// TwinCAT 3 PLC project RFID_lib
// Title: RFID_Sensor
// Company: Thomas More
// Author: Arno Joosen
// ProjectVersion: 0.0.4
// ProgramVersion: 3.1.4023.0
// libraries:
//   Buffer Lib, * (Thomas More)
//   RFID universal data interface TwinCAT, * (Turck)
//   Tc2_Standard, * (Beckhoff Automation GmbH)
//   Tc2_System, * (Beckhoff Automation GmbH)
//   Tc3_Module, * (Beckhoff Automation GmbH)
// project tree:
//   DUTs/ Read_State.TcDUT, RFID_Sensor.TcDUT, RFID_SensorState.TcDUT, RFID_Error.TcDUT, RFID_Tag_Data.TcDUT, Tag_UID.TcDUT, Wread_State.TcDUT
//   POUs/ ID_equal_to_ID.TcPOU, RFID_Sensor_Read.TcPOU, RFID_Sensor_Wread.TcPOU, RFID_Update.TcPOU
//   POUs/Read_Tag_Data/ RFID_Get_Bool.TcPOU, RFID_Get_Int.TcPOU, RFID_Get_Real.TcPOU, RFID_Get_String.TcPOU
//   POUs/Wread_Tag_Data/ RFID_Set_Bool.TcPOU, RFID_Set_Int.TcPOU, RFID_Set_Real.TcPOU, RFID_Set_String.TcPOU
//   Version/ Global_Version.TcGVL
// real-time tasks:
//   TASK PlcTask: cycle T#10ms, priority 20, ADS port 350
//   TASK PlcTask1: cycle T#10ms, priority 21, ADS port 351
//   TASK PlcTask2: cycle T#10ms, priority 22, ADS port 352
//   TASK PlcTask3: cycle T#10ms, priority 23, ADS port 353

// ---- DUTs/Read_State.TcDUT
{attribute 'qualified_only'}
{attribute 'strict'}
TYPE Read_State :
(
	Triggerd := 0,
	DataWritten := 1,
	Done := 2
)UINT;
END_TYPE

// ---- DUTs/RFID_Sensor.TcDUT
TYPE RFID_Sensor :
STRUCT
	Input AT %I* : CompactInput_t;
	Ouput AT %Q* : CompactOutput_t;
	
	Input_Buffer AT %I* : ARRAY[0..127] OF BYTE;
	Output_Buffer AT %Q* : ARRAY[0..127] OF BYTE;
	
	TxBuffer : ARRAY[0..127] OF BYTE;
	
	State : RFID_SensorState := RFID_SensorState.idel;
	ReadState : Read_State;
	WreadState : Wread_State;
	Pagina : UINT;
	CurrentTagData : RFID_Tag_Data;
END_STRUCT
END_TYPE

// ---- DUTs/RFID_SensorState.TcDUT
{attribute 'qualified_only'}
{attribute 'strict'}
TYPE RFID_SensorState :
(
	idel := 0,
	ReadTag := 1,
	WreadTag := 2,
	Error := 3
) UINT;
END_TYPE

// ---- DUTs/RFID_Error.TcDUT
{attribute 'qualified_only'}
{attribute 'strict'}
TYPE RFID_Error :
(
	None := 0,
	Not_Connected := 1,
	Time_Out := 2,
	Sesnor := 3
) UINT;
END_TYPE

// ---- DUTs/RFID_Tag_Data.TcDUT
TYPE RFID_Tag_Data :
STRUCT
	Data : ARRAY[0..127] OF BYTE;
	UID : Tag_UID;
	Layout : Buffer_Layout;
END_STRUCT
END_TYPE

// ---- DUTs/Tag_UID.TcDUT
TYPE Tag_UID : ARRAY[0..7] OF USINT; END_TYPE

// ---- DUTs/Wread_State.TcDUT
{attribute 'qualified_only'}
{attribute 'strict'}
TYPE Wread_State :
(
	Triggerd := 0,
	DataWritten := 1,
	Done := 2
);
END_TYPE

// ---- Version/Global_Version.TcGVL
{attribute 'TcGenerated'}
{attribute 'no-analysis'}
{attribute 'linkalways'}
// This function has been automatically generated from the project information.
VAR_GLOBAL CONSTANT
	{attribute 'const_non_replaced'}
	stLibVersion_RFID_Sensor : ST_LibVersion := (iMajor := 0, iMinor := 0, iBuild := 4, iRevision := 0, nFlags := 0, sVersion := '0.0.4');
END_VAR

// ---- POUs/ID_equal_to_ID.TcPOU
FUNCTION ID_equal_to_ID : BOOL
VAR_INPUT
	ID1 :  REFERENCE TO Tag_UID;
	ID2 :  REFERENCE TO Tag_UID;
END_VAR

VAR CONSTANT 
	TagSize : UINT := 8;
END_VAR

VAR
	i : UINT;
	TagEqual : BOOL := TRUE;
END_VAR

FOR i:=0 TO TagSize-1 BY 1 DO
	TagEqual := TagEqual AND ID1[i] = ID2[i];
	// TODO Stop for loop waneer niet gelijk
END_FOR

ID_equal_to_ID := TagEqual;

END_FUNCTION

// ---- POUs/Read_Tag_Data/RFID_Get_Bool.TcPOU
FUNCTION RFID_Get_Bool : Buffer_Error
VAR_INPUT
	Data : REFERENCE TO RFID_Tag_Data;
	Num : USINT; 
END_VAR
VAR_IN_OUT
	Out : BOOL;
END_VAR

RFID_Get_Bool := Get_Bool_From_Buffer(Num:= Num, 
									Layout:= Data.Layout, 
									Buffer:= Data.Data, 
									Out:= Out);

END_FUNCTION

// ---- POUs/Read_Tag_Data/RFID_Get_Int.TcPOU
FUNCTION RFID_Get_Int : Buffer_Error
VAR_INPUT
	Data : REFERENCE TO RFID_Tag_Data;
	Num : USINT; 
END_VAR
VAR_IN_OUT
	Out : INT;
END_VAR

RFID_Get_Int := Get_Int_From_Buffer(Num:= Num, 
									Layout:= Data.Layout, 
									Buffer:= Data.Data, 
									Out:= Out);

END_FUNCTION

// ---- POUs/Read_Tag_Data/RFID_Get_Real.TcPOU
FUNCTION RFID_Get_Real : Buffer_Error
VAR_INPUT
	Data : REFERENCE TO RFID_Tag_Data;
	Num : USINT; 
END_VAR
VAR_IN_OUT
	Out : REAL;
END_VAR

RFID_Get_Real := Get_Real_From_Buffer(Num:= Num, 
										Layout:= Data.Layout, 
										Buffer:= Data.Data, 
										Out:= Out);

END_FUNCTION

// ---- POUs/Read_Tag_Data/RFID_Get_String.TcPOU
FUNCTION RFID_Get_String : Buffer_Error
VAR_INPUT
	Data : REFERENCE TO RFID_Tag_Data;
	Num : USINT; 
END_VAR
VAR_IN_OUT
	Out : STRING[8];
END_VAR

RFID_Get_String := Get_String_From_Buffer(Num:= Num, 
											Layout:= Data.Layout, 
											Buffer:= Data.Data, 
											Out:= Out);

END_FUNCTION

// ---- POUs/RFID_Sensor_Read.TcPOU
FUNCTION RFID_Sensor_Read : bool
VAR_INPUT
	Layout : Buffer_Layout;
	P : UINT;
END_VAR
VAR_IN_OUT
	Sensor : RFID_Sensor;
END_VAR

IF (P < 64) AND (Sensor.State = RFID_SensorState.idel) THEN
	Sensor.State := RFID_SensorState.ReadTag;
	Sensor.ReadState := Read_State.Triggerd;
	Sensor.Pagina := P;
	Sensor.CurrentTagData.Layout := Layout;
END_IF

END_FUNCTION

// ---- POUs/RFID_Sensor_Wread.TcPOU
FUNCTION RFID_Sensor_Wread : BOOL
VAR_INPUT
	Data : REFERENCE TO RFID_Tag_Data;
	P : UINT;
END_VAR
VAR_IN_OUT
	Sensor : RFID_Sensor;
END_VAR

IF (P < 64) AND (Sensor.State = RFID_SensorState.idel) THEN
	Sensor.State := RFID_SensorState.WreadTag;
	Sensor.WreadState := Wread_State.Triggerd;
	Sensor.Pagina := P;
	Sensor.TxBuffer := Data.Data;
END_IF

END_FUNCTION

// ---- POUs/RFID_Update.TcPOU
FUNCTION_BLOCK RFID_Update
VAR_IN_OUT
	Sensor : RFID_Sensor;
END_VAR

VAR_OUTPUT
	Q : BOOL;
	Tag_Data : RFID_Tag_Data;
	Error : RFID_Error;
END_VAR

VAR
	TagFB: FB_Compact;
	Execute : BOOL;
	Abort : BOOL;
	TimeOut : UDINT := 1000000; 
	Command : COMMAND;
	Done : BOOL;
	Busy : BOOL;
	_Error : BOOL;
	Aborted : BOOL;
	ErrorID : ERROR;
	TagDetekt : BOOL;
	NotConekted : BOOL;
	LData : UINT;
	Adress : UDINT := 0;
	Length : UINT := 0;
	i : UINT;
	RxBuffer : ARRAY[0..127] OF BYTE;
END_VAR

CASE Sensor.State OF
	RFID_SensorState.idel:
		Command := 16#0;
		Execute := FALSE;
		Execute_TagFB();
	RFID_SensorState.ReadTag:
		Read_StateMachine();
		Execute_TagFB();
	RFID_SensorSTATE.WreadTag:
		Wread_StateMachine();
		Execute_TagFB();
END_CASE

IF NOT (Sensor.State = RFID_SensorState.Error) THEN
	Q := TagDetekt;
	IF TagDetekt THEN
		FOR i := 0 TO 7 BY 1 DO
			Sensor.CurrentTagData.UID[i] := Sensor.Input_Buffer[i];
		END_FOR
	END_IF
END_IF

IF _Error THEN
	Sensor.State := RFID_SensorState.Error;
	CASE ErrorID OF
		1:
			Error := RFID_Error.Time_Out;
		ELSE
			Error := RFID_Error.Sesnor;
	END_CASE
ELSIF NotConekted THEN
	Sensor.State := RFID_SensorState.Error;
	Error := RFID_Error.Not_Connected;
ELSE
	Error := RFID_Error.None;
	Tag_Data := Sensor.CurrentTagData;
END_IF

ACTION Execute_TagFB:
TagFB(
	xExecute:= Execute, // BOOL
	xAbort:= Abort, // BOOL
	udiTimeOut:= TimeOut, // UDINT
	xDone=> Done, // BOOL
	xBusy=> Busy, // BOOL
	xError=> _Error, // BOOL
	xAborted=> Aborted, // BOOL
	eCommand:= Command, /// COMMAND
		// This command wil be executed on xEcecute
	rStatusMapping:= Sensor.Input, // REFFERENCE TO CompactInput_t
		// input data of the compact module
	rControlMapping:= Sensor.Ouput, // REFEREANCE TO CompactOuput_t
		// output data of the compact module
	udiStartAddress:= Adress, // UDINT
		// the address defines the adress in the context of the command 
		// defined by the command code I.E. the adress of the data within the tag memory
	uiDataLength:= Length, // UINT
		// de length of data to be read or written or the size of the inventory response
	eErrorID=> ErrorID, // ERROR
	xTP=> TagDetekt, // BOOL
		// tag whithin the detection range
	xRWHeadNotConnected=> NotConekted, // BOOL
		// read/write had not connected
	uiDataRxLength=> LData,  // UINT
		// the length defines the legth in the context of the command 
		// defined by the command code I.E. the length of data to be read or written or the 
		// size of the inventory response
	pReadDataMapping:= Sensor.Input_Buffer, // POINTER TO BYTE
		// start adress of the input data i.e. input data of the read data module e.g.g ADR()
	pWriteDataMapping:= Sensor.Output_Buffer, // PONTER TO BYTE
		// start address of the ouput data i.e. ouput data of the write data module
	pDataTx:= Sensor.TxBuffer, // POINTER TO BYTE
		// buffer which contains the data to be written
	pDataRx:= RxBuffer // PINTER TO BYTE
		// buffer which stores the read data
);
END_ACTION

ACTION Read_StateMachine:
IF Sensor.ReadState = Read_State.Triggerd THEN
	Command := 16#2;
	Adress := Sensor.Pagina * 128;
	Length := 128;
	Sensor.ReadState := Read_State.DataWritten;
ELSIF Sensor.ReadState = Read_State.DataWritten THEN
	Execute := TRUE;
	IF Done AND NOT _Error THEN
		Sensor.ReadState := Read_State.Done;
	END_IF
ELSIF Sensor.ReadState = Read_State.Done THEN
	Execute := FALSE;
	Sensor.State := RFID_SensorState.idel;
	MEMCPY(destAddr:= ADR(Sensor.CurrentTagData.Data), srcAddr:= ADR(RxBuffer), n:= 128);
END_IF
END_ACTION

ACTION Wread_StateMachine:
IF Sensor.WreadState = Wread_State.Triggerd THEN
	Command := 16#4;
	Adress := Sensor.Pagina * 128;
	Length := 128;
	Sensor.WreadState := Wread_State.DataWritten;
ELSIF Sensor.WreadState = Wread_State.DataWritten THEN
	Execute := TRUE;
	IF Done AND NOT _Error THEN
		Sensor.WreadState := Wread_State.Done;
	END_IF
ELSIF Sensor.WreadState = Wread_State.Done THEN
	Execute := FALSE;
	Sensor.State := RFID_SensorState.idel;
END_IF
END_ACTION

END_FUNCTION_BLOCK

// ---- POUs/Wread_Tag_Data/RFID_Set_Bool.TcPOU
FUNCTION RFID_Set_Bool : Buffer_Error
VAR_INPUT
	In : BOOL;
	Num : USINT; 
END_VAR
VAR_IN_OUT
	Data : RFID_Tag_Data;
END_VAR

RFID_Set_Bool := Set_Bool_Fom_Buffer(In:= In, 
									Num:= Num, 
									Layout:= Data.Layout, 
									Buffer:= Data.Data);

END_FUNCTION

// ---- POUs/Wread_Tag_Data/RFID_Set_Int.TcPOU
FUNCTION RFID_Set_Int : Buffer_Error
VAR_INPUT
	In : INT;
	Num : USINT; 
END_VAR
VAR_IN_OUT
	Data : RFID_Tag_Data;
END_VAR

RFID_Set_Int := Set_Int_From_Buffer(In:= In, 
									Num:= Num, 
									Layout:= Data.Layout, 
									Buffer:= Data.Data);

END_FUNCTION

// ---- POUs/Wread_Tag_Data/RFID_Set_Real.TcPOU
FUNCTION RFID_Set_Real : Buffer_Error
VAR_INPUT
	In : REAL;
	Num : USINT; 
END_VAR
VAR_IN_OUT
	Data : RFID_Tag_Data;
END_VAR

RFID_Set_Real := Set_Real_From_Buffer(In:= In, 
										Num:= Num, 
										Layout:= Data.Layout, 
										Buffer:= Data.Data);

END_FUNCTION

// ---- POUs/Wread_Tag_Data/RFID_Set_String.TcPOU
FUNCTION RFID_Set_String : Buffer_Error
VAR_INPUT
	In : STRING[8];
	Num : USINT; 
END_VAR
VAR_IN_OUT
	Data : RFID_Tag_Data;
END_VAR

RFID_Set_String := Set_String_From_Buffer(In:= In, 
											Num:= Num, 
											Layout:= Data.Layout, 
											Buffer:= Data.Data);

END_FUNCTION
